{attribute 'GeneratedUsingTerminal: EK1122-0000-0018'}
{attribute addProperty BoxType "EK1122-0000-0018"}
{attribute addProperty Id "Beckhoff_EQ1xxxsub_EK1100EK1100_AB5A94672A_0001_EQ1008_0002_0016EQ1008_4201D0AB12A_0002_EQ1008_0002_0017EQ1008_4201D0AB12A_0003_EQ1008_0002_0018EQ1008_4201D0AB12A_0004_EQ1809_0022_0016EQ1809_FD7895E220A_0005_EQ1809_0022_0018EQ1809_FD7895E220"}
{attribute addProperty CRC "25569060"}
{attribute addProperty Size "78"}
TYPE Beckhoff_EQ1xxxEK1122_01862724 EXTENDS EK1122_AB5A9467 :
STRUCT
	{attribute addProperty Name "Beckhoff_EQ1xxxsub_EK1100"}
	Beckhoff_EQ1xxxsub_EK1100 : EK1100_AB5A9467;
	{attribute addProperty Name "A_0001_EQ1008_0002_0016"}
	A_0001_EQ1008_0002_0016 : EQ1008_4201D0AB;
	{attribute addProperty Name "A_0002_EQ1008_0002_0017"}
	A_0002_EQ1008_0002_0017 : EQ1008_4201D0AB;
	{attribute addProperty Name "A_0003_EQ1008_0002_0018"}
	A_0003_EQ1008_0002_0018 : EQ1008_4201D0AB;
	{attribute addProperty Name "A_0004_EQ1809_0022_0016"}
	A_0004_EQ1809_0022_0016 : EQ1809_FD7895E2;
	{attribute addProperty Name "A_0005_EQ1809_0022_0018"}
	A_0005_EQ1809_0022_0018 : EQ1809_FD7895E2;
END_STRUCT
END_TYPE

(* stored: Version 1.2.0.0, ProductVersion 3.1.4024.9
   DUT Beckhoff_EQ1xxxEK1122_01862724: Id {3eb215cc-3dc6-43df-9ccd-7f04c7f9b7d4} *)
